FUNCTION_BLOCK EL3062
VAR
	_io : EL3xx2_Data;
	{attribute addProperty Name "WcState"}
	_wcState : WcStateInputToggle;
	{attribute addProperty Name "Info data"}
	_infoData : InfoDataAds;
END_VAR

PROPERTY IO : REFERENCE TO EL3xx2_Data
GET
IO REF= _io;
END_GET
END_PROPERTY

PROPERTY WcState : REFERENCE TO WcStateInputToggle
GET
WcState REF= _wcState;
END_GET
END_PROPERTY

END_FUNCTION_BLOCK

(* stored: Version 1.1.0.1, ProductVersion 3.1.4024.9
   POU EL3062: Id {afa3c8cf-4bce-0fb0-3532-9f32597c2753}, SpecialFunc None
   Property IO: Id {7ff04361-95cc-0329-0ae4-acad004f08a6}
   Get Get: Id {fac19fb3-63f9-032b-244e-83107e3a9ecc}
   Property WcState: Id {a408c1b7-270b-0652-3f72-7354c7428793}
   Get Get: Id {b7d3170e-3194-01bb-2885-c0bb68b996be} *)
